// TIA Portal V20 export
FUNCTION_BLOCK "zPMC_FaultWord"   // FB231, LAD
// stored: MemoryReserve 100, Namespace CITI_Logic, SetENOAutomatically false
   VAR_OUTPUT
      TMP_PMC_FaultIndex : Int;
   END_VAR
   VAR_IN_OUT
      FaultWords : Array[0..499] of Word;
   END_VAR
   VAR
      sFaultWords : Array[0..499] of Word;
      sDestArray : Array[1..8000] of Bool;
   END_VAR
   VAR_TEMP
      tInitializeFaults : Word;
      tIndex : Int;
   END_VAR
BEGIN

REGION Network 1: Initialize fault words
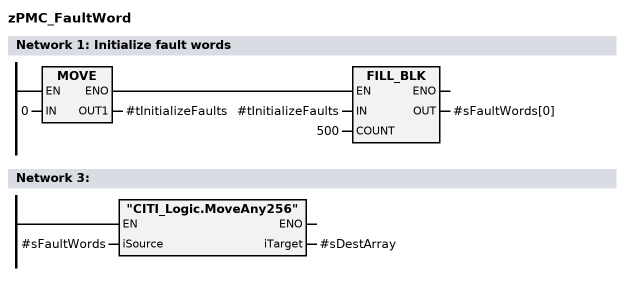
   RUNG wire#powerrail
      Move(in := 0, out1 => #tInitializeFaults)
      FillBlockI(in := #tInitializeFaults, count := 500, out => #sFaultWords[0])
   END_RUNG
   // the same network as SCL:
   #tInitializeFaults := 0;
   FILL_BLK(IN := #tInitializeFaults, COUNT := 500, OUT => #sFaultWords[0]);
END_REGION

REGION Network 2 (SCL): Swap byte order
   FOR #tIndex := 0 TO 499 DO
       // Statement section FOR
       // 
       #sFaultWords[#tIndex]:= SWAP_WORD(#FaultWords[#tIndex]);

       ;
   END_FOR;
END_REGION

REGION Network 3
   RUNG wire#powerrail
      "CITI_Logic.MoveAny256"(iSource := #sFaultWords, iTarget => #sDestArray)
   END_RUNG
   // the same network as SCL:
   "CITI_Logic.MoveAny256"(iSource := #sFaultWords, iTarget => #sDestArray);
END_REGION

REGION Network 4 (SCL)
   FOR #tIndex := 1 TO 8000 DO
       // Statement section FOR
       // 

       IF #sDestArray[#tIndex] = TRUE THEN
           // Statement section IF
           // 
           #TMP_PMC_FaultIndex := #tIndex;


           EXIT;


           ;
       END_IF;




       ;
   END_FOR;
END_REGION
END_FUNCTION_BLOCK
